// TIA Portal V19 export
TYPE "typePressureGuageRs485ControlNodeCommands"
TITLE = LBC_typeAnalogOutputControlNodeCommands
// Control Node Wapper commands
// stored: Access Published
   STRUCT
      simulation { ExternalAccessible := 'False'; ExternalVisible := 'False'; ExternalWritable := 'False'} : Bool;   // Manual mode parameters for axis control interface
      simulatedAnalogValue { ExternalAccessible := 'False'; ExternalVisible := 'False'; ExternalWritable := 'False'} : Int;   // Input process value for scaling from simulated process
      reset { ExternalAccessible := 'False'; ExternalVisible := 'False'; ExternalWritable := 'False'} : Bool;   // Manual mode parameters for axis control interface
      quality { ExternalAccessible := 'False'; ExternalVisible := 'False'; ExternalWritable := 'False'} : Bool := true;   // Manual mode parameters for axis control interface
   END_STRUCT;
END_TYPE
